PROGRAM CirculationPumpEx
VAR
	fbHVACCirculationPumpEx: FB_HVACCirculationPumpEx;
	eDataSecurityType: E_HVACDataSecurityType := E_HVACDataSecurityType.eHVACDataSecurityType_Idle;
	bSetDefault: BOOL;
	bEnable: BOOL := TRUE;
	bExternal: BOOL;
	eCtrlModeActuator: E_HVACActuatorMode;
	rOutsideTemp: REAL;
	rValvePosition: REAL;
	bFeedbPump: BOOL := TRUE;
	bPumpProtec: BOOL := TRUE;
	bManSwitch: BOOL := TRUE;
	bCtrlVoltage: BOOL := TRUE;
	bReset: BOOL;
	bPump: BOOL;
	byState: BYTE;
	bReqExternal: BOOL;
	bReqOutsideTemp: BOOL;
	bReqValve: BOOL;
	bStateManSwitch: BOOL;
	udiSecRT_StopDelay: UDINT;
	udiSecRT_FeedbPumpDelay: UDINT;
	eStateModeActuator: Tc2_HVAC.E_HVACActuatorMode;
	bError: BOOL;
	byError: BYTE;
	bErrorPumpProtec: BOOL;
	bErrorFeedb: BOOL;
	bInvalidParameter: BOOL;
	udiSecStopDelay: UDINT;
	udiSecFeedbPumpDelay: UDINT;
	rOutsideTempHighLimit: REAL;
	rOutsideTempLowLimit: REAL;
	rValvePositionLimitOn: REAL;
	rValvePositionLimitOff: REAL;
	eReqPump: E_HVACReqPump;
END_VAR

fbHVACCirculationPumpEx(
	eDataSecurityType:=eDataSecurityType, 
	bSetDefault:=bSetDefault, 
	bEnable:=bEnable, 
	bExternal:=bExternal, 
	eCtrlModeActuator:=eCtrlModeActuator, 
	rOutsideTemp:=rOutsideTemp, 
	rValvePosition:=rValvePosition, 
	bFeedbPump:=bFeedbPump, 
	bPumpProtec:=bPumpProtec, 
	bManSwitch:=bManSwitch, 
	bCtrlVoltage:=bCtrlVoltage, 
	bReset:=bReset, 
	bPump=>bPump, 
	byState=>byState, 
	bReqExternal=>bReqExternal, 
	bReqOutsideTemp=>bReqOutsideTemp, 
	bReqValve=>bReqValve, 
	bStateManSwitch=>bStateManSwitch, 
	udiSecRT_StopDelay=>udiSecRT_StopDelay, 
	udiSecRT_FeedbPumpDelay=>udiSecRT_FeedbPumpDelay, 
	eStateModeActuator=>eStateModeActuator, 
	bError=>bError, 
	byError=>byError, 
	bErrorPumpProtec=>bErrorPumpProtec, 
	bErrorFeedb=>bErrorFeedb, 
	bInvalidParameter=>bInvalidParameter, 
	udiSecStopDelay:=udiSecStopDelay, 
	udiSecFeedbPumpDelay:=udiSecFeedbPumpDelay, 
	rOutsideTempHighLimit:=rOutsideTempHighLimit, 
	rOutsideTempLowLimit:=rOutsideTempLowLimit, 
	rValvePositionLimitOn:=rValvePositionLimitOn, 
	rValvePositionLimitOff:=rValvePositionLimitOff, 
	eReqPump:=eReqPump);

END_PROGRAM

(* stored: Version 1.1.0.1, ProductVersion 3.1.4024.4
   POU CirculationPumpEx: Id {aabfa980-3fe3-4242-a1c7-fc502b27c3e6}, SpecialFunc None *)
